TYPE RemoteFeedbackLeica :
STRUCT
	x : REAL;
	y : REAL;
	z : REAL;
	q0 : REAL;
	q1 : REAL;
	q2 : REAL;
	q3 : REAL;
END_STRUCT
END_TYPE

(* stored: Version 1.1.0.1, ProductVersion 3.1.4020.12
   DUT RemoteFeedbackLeica: Id {753df343-d8a4-4be5-aa7a-1ee5fc5c7942} *)
